FUNCTION_BLOCK REPORT_IF_GREATER
  {SET_ATTRIBUTE(OpcUa, SERVICE)}
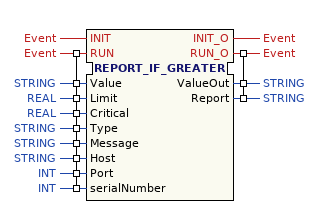
  EVENT_INPUT
    INIT;
    RUN WITH Value, Limit, Critical, Type, Message, Host, Port, serialNumber; {SET_ATTRIBUTE(OpcUa, Method)}
  END_EVENT
  EVENT_OUTPUT
    INIT_O;
    RUN_O WITH ValueOut, Report;
  END_EVENT
  VAR_INPUT
    Value : STRING; {SET_ATTRIBUTE(OpcUa, Variable.RUN)}
    Limit : REAL; {SET_ATTRIBUTE(OpcUa, Variable.RUN)}
    Critical : REAL; {SET_ATTRIBUTE(OpcUa, Variable.RUN)}
    Type : STRING; {SET_ATTRIBUTE(OpcUa, Variable.RUN)}
    Message : STRING; {SET_ATTRIBUTE(OpcUa, Variable.RUN)}
    Host : STRING; {SET_ATTRIBUTE(OpcUa, Variable.RUN)}
    Port : INT; {SET_ATTRIBUTE(OpcUa, Variable.RUN)}
    serialNumber : INT; {SET_ATTRIBUTE(OpcUa, Variable.RUN)}
  END_VAR
  VAR_OUTPUT
    ValueOut : STRING; {SET_ATTRIBUTE(OpcUa, Variable.RUN)}
    Report : STRING; {SET_ATTRIBUTE(OpcUa, Variable.RUN)}
  END_VAR
END_FUNCTION_BLOCK
